FUNCTION_BLOCK FB_ADS_CleanAxis EXTENDS FB_AdsBlockBase
VAR
  // ---------------------------------
  // ADS interface block specific
  sO_Message            : ST_ADS_MSG_IF;    (*Messaging*)

  bI_FaultAck           : BOOL := FALSE;

  (*Manual Move, only possible when in maintenance and manual mode*)
  bI_ManualMove         : BOOL := FALSE;  (*Active as long as true*)
  bO_ManualMoveCanEx    : BOOL := FALSE;
  bO_ManualMovekExec    : BOOL := FALSE;
  fI_ManualTargetPos    : REAL := 0.0;

  (*Current axis position*)
  sO_AxisPosition       : ST_VAR_OUT_REAL;

  wO_ErrorCode          : WORD;
  bO_Busy               : BOOL;
  bO_Ready              : BOOL;
  bO_Error              : BOOL;
END_VAR

VAR PERSISTENT
  nR_Pattern            : UDINT;  (*check pattern for rem validity*)
END_VAR

METHOD config
VAR_INPUT
  aName               : STRING;
  sAxisPositionUnit   : STRING;  
  fAxisPositionMin    : REAL;  
  fAxisPositionMax    : REAL;  
END_VAR
aO_Name                  := aName;

sO_AxisPosition.bC_Exist := TRUE; 
sO_AxisPosition.aC_Unit  := sAxisPositionUnit; 
sO_AxisPosition.fC_Min   := fAxisPositionMin; 
sO_AxisPosition.fC_Max   := fAxisPositionMax; 

(*OPC-UA: EngineeringUnits*)
sO_AxisPosition.nC_EngineeringUnits := 5066068;  (*[mm]*)
END_METHOD

METHOD PROTECTED initRemVar
VAR_INPUT
END_VAR
(*load default initial values if pattern was invalid*)
IF nR_Pattern <> 16#ABCD THEN
  ;
ELSE  
  nR_Pattern      := 16#ABCD;
END_IF

(*Init values*)
END_METHOD

METHOD ResetCommands : BOOL
VAR_INPUT
END_VAR
bI_ManualMove := FALSE;
END_METHOD

METHOD setFeedback
VAR_INPUT
  bManualMoveCanEx         : BOOL; 
  bManualMovekExec         : BOOL;  

  fAxisPositionVal         : REAL;  

  wErrorCode               : WORD; 
  bBusy                    : BOOL; 
  bReady                   : BOOL; 
  bError                   : BOOL; 
END_VAR
bO_ManualMoveCanEx         := bManualMoveCanEx;
bO_ManualMovekExec         := bManualMovekExec;

sO_AxisPosition.fO_Val     := fAxisPositionVal;

wO_ErrorCode               := wErrorCode;
bO_Busy                    := bBusy;
bO_Ready                   := bReady;
bO_Error                   := bError;
END_METHOD

(*
  Setup constant ADS Block definitions.
  HOWTO: in abstract implmentation call
      init(aVersion:=, aType:=, nType:=, eLayer:=);
*)
METHOD  setup
init( aVersion := '01.00.01'
    , aType    := 'CleanAxis'
    , nType    := eMa_BLK_MACHINE
    , eLayer   := E_AdsLayer.Structural);
END_METHOD

PROPERTY sMsgInterface : POINTER TO ST_ADS_MSG_IF
GET
sMsgInterface := ADR(sO_Message);
END_GET
END_PROPERTY

END_FUNCTION_BLOCK

(* stored: Version 1.1.0.1, ProductVersion 3.1.4024.11
   POU FB_ADS_CleanAxis: Id {e81195e2-8818-4f5a-9a27-42b320bc7d25}, SpecialFunc None
   Method config: Id {602858fe-2d47-42ed-b907-702dfdb24639}
   Method initRemVar: Id {ec2a8444-5ba7-4906-93b7-26c86a7e3c78}
   Method ResetCommands: Id {e3c86916-a8f3-41c7-9565-d69df5982317}
   Method setFeedback: Id {808e9ee2-01fc-4620-b610-7daa8bbe91ac}
   Method setup: Id {480b63e7-c4e5-483a-b879-6d3a3d0139cb}
   Property sMsgInterface: Id {cb86ee4f-a925-4f0a-a2ca-82963da655b0}
   Get Get: Id {037e6469-2d88-4619-b074-485e9444d141} *)
